{attribute 'linkalways'} 
{attribute 'no_explicit_call' := 'This FB is a CLASS and must be accessed using methods or properties'}
{attribute 'enable_dynamic_creation'}
FUNCTION_BLOCK PUBLIC BasicDigitalOutput IMPLEMENTS I_DigitalOutput
VAR
	output AT %Q* : BOOL;
	inverted : BOOL;
END_VAR

METHOD FB_init : BOOL
VAR_INPUT
	bInitRetains : BOOL; // if TRUE, the retain variables are initialized (warm start / cold start)
	bInCopyCode : BOOL;  // if TRUE, the instance afterwards gets moved into the copy code (online change)
	inverted : BOOL;
END_VAR
THIS^.inverted := inverted;
END_METHOD

{attribute 'monitoring' := 'call'}
PROPERTY PUBLIC State : BOOL
GET // PUBLIC
State := output XOR inverted;
END_GET
SET // PUBLIC
output := State XOR inverted;
END_SET
END_PROPERTY

END_FUNCTION_BLOCK

(* stored: Version 1.1.0.1, ProductVersion 3.1.4024.12
   POU BasicDigitalOutput: Id {f027e06b-59a5-4ebb-b9f8-6ec4a5c0ac66}, SpecialFunc None
   Method FB_init: Id {c086133b-732b-412d-8b23-1d473bf6dd52}
   Property State: Id {f0765697-fa40-4e8a-821d-685c010b2db3}
   Get Get: Id {9b741276-af2e-48a4-be51-3e3e011beff7}
   Set Set: Id {7bfd0bb2-6c59-4c5f-b904-bee495afa607} *)
